FUNCTION_BLOCK MixerLogic_HMI (* Service Interface Function Block Type *)
  (* Standard: 61499-2 *)
  (* Version 0.0, 6/15/2026, Schneider Electric, template *)
  PACKAGE SE.Nereda;
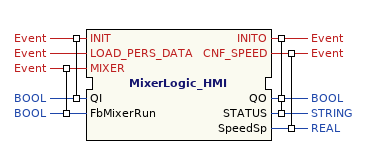
  EVENT_INPUT
    INIT WITH QI;
    LOAD_PERS_DATA;
    MIXER WITH FbMixerRun;
  END_EVENT
  EVENT_OUTPUT
    INITO WITH QO, STATUS;
    CNF_SPEED WITH SpeedSp;
  END_EVENT
  VAR_INPUT
    QI : BOOL;
    FbMixerRun : BOOL;
  END_VAR
  VAR_OUTPUT
    QO : BOOL; (* Event Output Qualifier *)
    STATUS : STRING; (* Service Status *)
    SpeedSp : REAL;
  END_VAR
  SERVICE /
    SEQUENCE 
    END_SEQUENCE
  END_SERVICE
END_FUNCTION_BLOCK
